{attribute 'GeneratedUsingTerminal: EK1200-1388-0000'}
{attribute addProperty VendorId "#x00000002"}
{attribute addProperty BoxType "EK1200-1388-0000"}
{attribute addProperty Description "EK1200-5000 EtherCAT Power supply (2A E-Bus)"}
{attribute addProperty Physics "YK"}
{attribute addProperty Id "EK1200"}
{attribute addProperty CRC "20777801"}
{attribute addProperty Size "0"}
TYPE EK1200_013D0B49 EXTENDS TcoIo.EtcSlaveBoxBase_77A0E4A7 :
STRUCT
END_STRUCT
END_TYPE

(* stored: Version 1.2.0.0
   DUT EK1200_013D0B49: Id {c6d55c21-45d4-49c6-b591-e46141dc51fa} *)
